Xinje XDPPro project, PLC1: XDH-60T4 (software 3.7.18 2024-11-27)

PROGRAM 梯形图

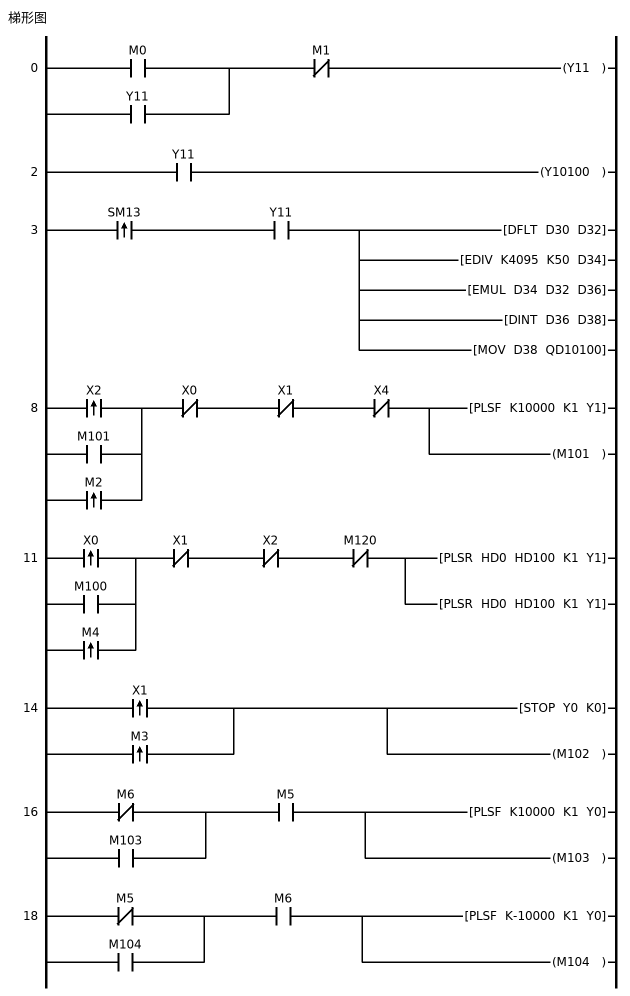
LD     M0
OR     Y11
ANI    M1
OUT    Y11
LD     Y11
OUT    Y10100
LDP    SM13
AND    Y11
DFLT   D30 D32
EDIV   K4095 K50 D34
EMUL   D34 D32 D36
DINT   D36 D38
MOV    D38 QD10100
LDP    X2
OR     M101
ORP    M2
ANI    X0
ANI    X1
ANI    X4
PLSF   K10000 K1 Y1
OUT    M101
LDP    X0
OR     M100
ORP    M4
ANI    X1
ANI    X2
ANI    M120
PLSR   HD0 HD100 K1 Y1
PLSR   HD0 HD100 K1 Y1
LDP    X1
ORP    M3
STOP   Y0 K0
OUT    M102
LDI    M6
OR     M103
AND    M5
PLSF   K10000 K1 Y0
OUT    M103
LDI    M5
OR     M104
AND    M6
PLSF   K-10000 K1 Y0
OUT    M104
Xinje XDPPro project, PLC2: XDH-60T4 (software 3.7.18 2024-11-27)

PROGRAM 梯形图

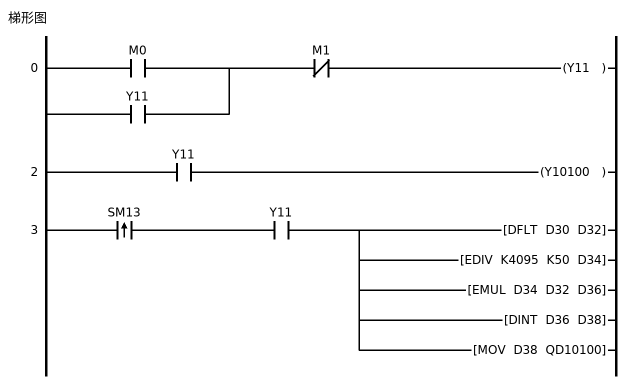
LD     M0
OR     Y11
ANI    M1
OUT    Y11
LD     Y11
OUT    Y10100
LDP    SM13
AND    Y11
DFLT   D30 D32
EDIV   K4095 K50 D34
EMUL   D34 D32 D36
DINT   D36 D38
MOV    D38 QD10100